{attribute 'qualified_only'}
VAR_GLOBAL
	Count	:	CTU;
END_VAR

(* stored: Version 1.1.0.1, ProductVersion 3.1.4024.9
   GVL CountUp: Id {d66f1d73-a710-4ebc-927f-e3685582c1c1} *)
